Staubli VAL3: newCommand.pgx

public program newCommand(pointRx& x_pPointCommand[])
  local num l_nNowPointPos[6]
  local num l_nNum
  local num l_nPointAccel[6]
  local num l_nPointPos[6]
  local num l_nPointVel[6]
  local num l_ndPointPos[6]
  local num l_nPostureTemp[3]
begin

  //===================== 每4ms更新机器人的位置指令（根据上一次采集的数据对下一次的运动产生修正） ====================

  while true

    //将机器人当前与理想的笛卡尔位置赋值给数组变量，便于程序操作（可采用参数传递操作数据）
    l_nNowPointPos[0]=pNowPointPos.trsf.x/1000
    l_nNowPointPos[1]=pNowPointPos.trsf.y/1000
    l_nNowPointPos[2]=pNowPointPos.trsf.z/1000
    l_nNowPointPos[3]=pNowPointPos.trsf.rx
    l_nNowPointPos[4]=pNowPointPos.trsf.ry
    l_nNowPointPos[5]=pNowPointPos.trsf.rz

    l_ndPointPos[0]=pdPointPos.trsf.x/1000
    l_ndPointPos[1]=pdPointPos.trsf.y/1000
    l_ndPointPos[2]=pdPointPos.trsf.z/1000
    l_ndPointPos[3]=pdPointPos.trsf.rx
    l_ndPointPos[4]=pdPointPos.trsf.ry
    l_ndPointPos[5]=pdPointPos.trsf.rz


    //---------- 基于阻抗/other模型，求出机器人下一条位置指令的误差修正量（注意单位换算） ----------
    //求加速度（位置+姿态）
    for l_nNum=0 to 2
      l_nPointAccel[l_nNum]=ndPointAccel[l_nNum]+1/nMass[l_nNum,l_nNum]*((ndForceTorque[l_nNum]-nForceTorque[l_nNum])-nDamp[l_nNum,l_nNum]*(nNowPointVel[l_nNum]-ndPointVel[l_nNum])/1000-nStiffness[l_nNum,l_nNum]*(l_nNowPointPos[l_nNum]-l_ndPointPos[l_nNum]))
      l_nPostureTemp[l_nNum]=1/nMass[l_nNum+3,l_nNum+3]*((ndForceTorque[l_nNum+3]-nForceTorque[l_nNum+3])-nDamp[l_nNum+3,l_nNum+3]*(nNowPointVel[l_nNum+3]-ndPointVel[l_nNum+3])-nStiffness[l_nNum+3,l_nNum+3]*(l_nNowPointPos[l_nNum+3]-l_ndPointPos[l_nNum+3]))
      l_nPointAccel[l_nNum+3]=ndPointAccel[l_nNum+3]+l_nPostureTemp[l_nNum]
    endFor

    //求速度（位置+姿态）
    for l_nNum=0 to 2
      l_nPointVel[l_nNum]=nNowPointVel[l_nNum]/1000+l_nPointAccel[l_nNum]*0.004
      l_nPointVel[l_nNum+3]=nNowPointVel[l_nNum+3]+l_nPointAccel[l_nNum+3]*0.004
    endFor

    //求位置指令（位置+姿态）（转换成笛卡儿坐标点类型（单位）并输出）
    for l_nNum=0 to 2
      l_nPointPos[l_nNum]=l_nNowPointPos[l_nNum]*1000+l_nPointVel[l_nNum]*0.004*1000
      l_nPointPos[l_nNum+3]=l_nNowPointPos[l_nNum+3]+l_nPointVel[l_nNum+3]*0.004
    endFor

    x_pPointCommand.trsf.x=l_nPointPos[0]
    x_pPointCommand.trsf.y=l_nPointPos[1]
    x_pPointCommand.trsf.z=l_nPointPos[2]
    x_pPointCommand.trsf.rx=l_nPointPos[3]
    x_pPointCommand.trsf.ry=l_nPointPos[4]
    x_pPointCommand.trsf.rz=l_nPointPos[5]

    //目前只修正机器人的位置部分,姿态部分暂时保持不变
//    x_pPointCommand.trsf.rx=pNowPointPos.trsf.rx
//    x_pPointCommand.trsf.ry=pNowPointPos.trsf.ry
//    x_pPointCommand.trsf.rz=pNowPointPos.trsf.rz


    //强制结束当前任务，进入下一次sequence循环
    delay(0.0)

  endWhile

end
